// TIA Portal V20 export
TYPE "LER_typeBrakeTestUnitInterface"
// stored: Access Published
   STRUCT
      commands { S7_SetPoint := 'True'} : "LER_typeBrakeTestUnitCommands";
      monitoring { ExternalWritable := 'False'; S7_SetPoint := 'True'} : "LER_typeBrakeTestUnitMonitoring";
   END_STRUCT;
END_TYPE
